FUNCTION_BLOCK DelayedAddCommand EXTENDS AddCommand
VAR
	_tonDelay		: TON := (PT:=T#4s);
END_VAR

METHOD PUBLIC Abort
SUPER^.Abort();

// Reset Input for next start
_tonDelay(IN:=stHandshake.bBusy);
END_METHOD

METHOD PROTECTED CalculateProgress
IF stHandshake.nResultCode = E_CommandResultCode.Done THEN
	stHandshake.nProgress := 100;
ELSE
	stHandshake.nProgress := REAL_TO_UINT(100.0 / TIME_TO_REAL(_tonDelay.PT) * TIME_TO_REAL(_tonDelay.ET));
END_IF
END_METHOD

METHOD PROTECTED Done
SUPER^.Done();

// Reset Input for next start
_tonDelay(IN:=stHandshake.bBusy);
END_METHOD

METHOD PROTECTED Task : BOOL
VAR_INPUT
	Init 	: BOOL;		// True the first time the Task is called after Execute is started
END_VAR
_tonDelay(IN:=stHandshake.bBusy);

IF _tonDelay.Q THEN
	// Execute base Task in AddCommand for Addition
	Task := SUPER^.Task(Init);
END_IF
END_METHOD

END_FUNCTION_BLOCK

(* stored: Version 1.1.0.1, ProductVersion 3.1.4022.10
   POU DelayedAddCommand: Id {65b2ca40-9e7e-4cdc-82b9-f7b2c503faa2}, SpecialFunc None
   Method Abort: Id {5607005d-a3e2-4a0d-8acf-89dd886f9689}
   Method CalculateProgress: Id {5cea9727-992d-40c4-9429-66e19c9b7a56}
   Method Done: Id {d3f67563-493c-480a-88ee-d8edb11f7e53}
   Method Task: Id {7c566ce4-fa9b-444f-bb18-8e5071761b78} *)
